{attribute addProperty BoxType "EL6201-0000-0017"}
{attribute addProperty Id "Slave_27A_DO0BIT10.125209Slave_27A_DO1BIT10.125210Slave_27A_DO2BIT10.125211Slave_27A_DO3BIT10.125212Slave_27B_DO0BIT10.125213Slave_27B_DO1BIT10.125214Slave_27B_DO2BIT10.125215Slave_27B_DO3BIT10.125216"}
{attribute addProperty CRC "4010556204"}
{attribute addProperty SizeInBites "8"}
{attribute addProperty SizeInBytes "1"}
TYPE Slave_27_Outputs_EF0C3B2C :
STRUCT
	{attribute addProperty Name "Slave_27A_DO0"}
	Slave_27A_DO0 : BIT;
	{attribute addProperty Name "Slave_27A_DO1"}
	Slave_27A_DO1 : BIT;
	{attribute addProperty Name "Slave_27A_DO2"}
	Slave_27A_DO2 : BIT;
	{attribute addProperty Name "Slave_27A_DO3"}
	Slave_27A_DO3 : BIT;
	{attribute addProperty Name "Slave_27B_DO0"}
	Slave_27B_DO0 : BIT;
	{attribute addProperty Name "Slave_27B_DO1"}
	Slave_27B_DO1 : BIT;
	{attribute addProperty Name "Slave_27B_DO2"}
	Slave_27B_DO2 : BIT;
	{attribute addProperty Name "Slave_27B_DO3"}
	Slave_27B_DO3 : BIT;
END_STRUCT
END_TYPE

(* stored: Version 1.2.0.0, ProductVersion 3.1.4024.9
   DUT Slave_27_Outputs_EF0C3B2C: Id {9531b13c-f6a1-46a8-8531-15ad7eba6829} *)
